FUNCTION_BLOCK DT2DT
  {SET_ATTRIBUTE(OpcUa, SERVICE)}
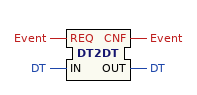
  EVENT_INPUT
    REQ;
  END_EVENT
  EVENT_OUTPUT
    CNF;
  END_EVENT
  VAR_INPUT
    IN : DT;
  END_VAR
  VAR_OUTPUT
    OUT : DT;
  END_VAR
END_FUNCTION_BLOCK
